TYPE E_ALM_PTS :
(
	PaperTransport 				:= 1,
	ModeParameter 				:= 2,
	TurnTableConfigMissmatch	:= 3,
	MAX_E_ALM_PTS
);
END_TYPE

(* stored: Version 1.1.0.1, ProductVersion 3.1.0.25
   DUT E_ALM_PTS: Id {054d011f-4a84-48e4-ba08-1819064b2746} *)
